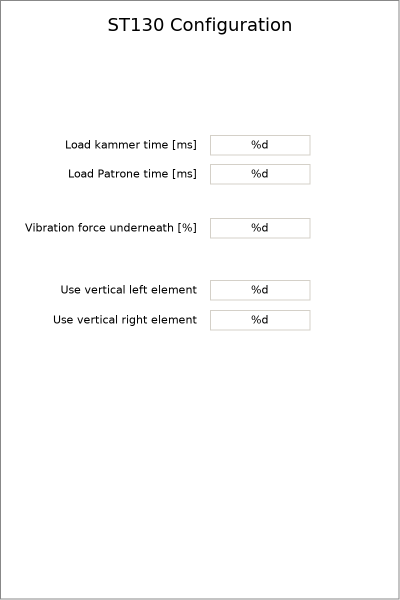
VISUALIZATION VISU_Recipe_ST130  // 400x600
    Label (0,5 400x40), "ST130 Configuration"
    Label (0,280 200x20), "Use vertical left element"
    Label (0,310 200x20), "Use vertical right element"
    Textfield (210,280 100x20), "%d", text variable: _20_AUTO.recipe.st130.xUseVerLeft
        OnMouseDown: write the text variable via Default
    Textfield (210,310 100x20), "%d", text variable: _20_AUTO.recipe.st130.xUseVerRight
        OnMouseDown: write the text variable via Default
    Label (0,135 200x20), "Load kammer time [ms]"
    Textfield (210,135 100x20), "%d", text variable: _20_AUTO.recipe.st130.diLoadKammer_ms
        OnMouseDown: write the text variable via Default
    Label (0,164 200x20), "Load Patrone time [ms]"
    Textfield (210,164 100x20), "%d", text variable: _20_AUTO.recipe.st130.diLoadPatrone_ms
        OnMouseDown: write the text variable via Default
    Label (0,218 200x20), "Vibration force underneath [%]"
    Textfield (210,218 100x20), "%d", text variable: _20_AUTO.recipe.st130.uiVibroUnderneath
        OnMouseDown: write the text variable via Default
END_VISUALIZATION

(* stored: Version 1.1.0.1, ProductVersion 3.1.4024.6
   Visu VISU_Recipe_ST130: Id {b4fd223c-2d77-4200-a2b5-41a74bab9ab5} *)
